FUNCTION PakcML_TO_TIME : ULINT
VAR_INPUT
	PackMLTime	:	ARRAY[0..6] OF DINT;
END_VAR
VAR
	nYear: DINT;
	nMonth:DINT;
	nDay:DINT;
	nHour:DINT;
	nMinute: DINT;
	nSecond: DINT;
	nMiliSecond:DINT;
	uiMsCount: INT;
	nResult : ULINT;
END_VAR

nYear := PackMLTime[0];
nMonth := PackMLTime[1];
nDay := PackMLTime[2];
nHour := PackMLTime[3];
nMinute := PackMLTime[4];
nSecond := PackMLTime[5];
nMiliSecond := PackMLTime[6];

FOR uiMsCount := 1 TO 12 DO
	nResult := nResult + daysInMonth(nYear := DINT_TO_INT(nYear),nMonth:=uiMsCount);
END_FOR

nResult := (nResult *24 + nHour)*60+nMinute;
nResult := nResult * 60 + nSecond;
nResult := nResult*1000 + nMiliSecond;

END_FUNCTION

(* stored: Version 1.1.0.1, ProductVersion 3.1.4024.11
   POU PakcML_TO_TIME: Id {9505d381-e609-4b89-88f3-042c532762a2}, SpecialFunc None *)
